{attribute 'linkalways'} 
{attribute 'no_explicit_call' := 'This FB is a CLASS and must be accessed using methods or properties'}
{attribute 'enable_dynamic_creation'}
FUNCTION_BLOCK _GVSP_PIXEL_FORMAT EXTENDS StructuredDatatypeBase
VAR
	localData : GVSP_PIXEL_FORMAT;
	activeData : REFERENCE TO GVSP_PIXEL_FORMAT REF= localData;
    _Color : _BYTE(localdata.Color);
    _EffectivePixelSize : _BYTE(localdata.EffectivePixelSize);
    _Id : _UINT(localdata.Id);
END_VAR

PROPERTY PUBLIC Address : PVOID
GET
Address := ADR(activeData);
END_GET
END_PROPERTY

METHOD PUBLIC ClearReference
VAR_INPUT
END_VAR
activeData REF= localData;
SetMemberReference();
END_METHOD

METHOD PUBLIC Clone : I_Datatype
VAR
    pClone : POINTER TO _GVSP_PIXEL_FORMAT;
END_VAR
pClone := __NEW(_GVSP_PIXEL_FORMAT());
pClone^.Value := Value;
Clone := pClone^;
END_METHOD

PROPERTY PUBLIC Color : REFERENCE TO _BYTE
GET
Color REF= _Color;
END_GET
END_PROPERTY

PROPERTY PUBLIC EffectivePixelSize : REFERENCE TO _BYTE
GET
EffectivePixelSize REF= _EffectivePixelSize;
END_GET
END_PROPERTY

METHOD FB_init : BOOL
VAR_INPUT
	bInitRetains : BOOL; // if TRUE, the retain variables are initialized (warm start / cold start)
	bInCopyCode : BOOL;  // if TRUE, the instance afterwards gets moved into the copy code (online change)
END_VAR
SetMemberReference();
AddMember('Color', _Color);
AddMember('EffectivePixelSize', _EffectivePixelSize);
AddMember('Id', _Id);
END_METHOD

PROPERTY PUBLIC Id : REFERENCE TO _UINT
GET
Id REF= _Id;
END_GET
END_PROPERTY

PROPERTY PUBLIC Identifier : T_MAXSTRING
GET
Identifier := 'GVSP_PIXEL_FORMAT';
END_GET
END_PROPERTY

METHOD PUBLIC MakeReferenceTo
VAR_INPUT
	ReferenceTarget : REFERENCE TO GVSP_PIXEL_FORMAT;
END_VAR
activeData REF= ReferenceTarget;
SetMemberReference();
END_METHOD

METHOD PROTECTED SetMemberReference
VAR_INPUT
END_VAR
_Color.MakeReferenceTo(activeData.Color);
_EffectivePixelSize.MakeReferenceTo(activeData.EffectivePixelSize);
_Id.MakeReferenceTo(activeData.Id);
END_METHOD

PROPERTY PUBLIC Size : UDINT
GET
Size := SIZEOF(activeData);
END_GET
END_PROPERTY

METHOD TryMakeReferenceTo : BOOL
VAR_INPUT
	Target : I_Datatype;
END_VAR
VAR
	targetAsStruct : I_StructuredDatatype;
	pTargetData : POINTER TO GVSP_PIXEL_FORMAT;
END_VAR
IF NOT Target.TryResolveAsStructuredDatatype(targetAsStruct) THEN
	RETURN;
END_IF

IF NOT (targetAsStruct.Identifier = Identifier) THEN
	RETURN;
END_IF

pTargetData := Target.Address;
activeData REF= pTargetData^;
SetMemberReference();
TryMakeReferenceTo := TRUE;
END_METHOD

PROPERTY PUBLIC Value : REFERENCE TO GVSP_PIXEL_FORMAT
GET
Value REF= activeData;
END_GET
END_PROPERTY

END_FUNCTION_BLOCK

(* stored: Version 1.1.0.1, ProductVersion 3.1.4024.13
   POU _GVSP_PIXEL_FORMAT: Id {a116f94a-4213-08f9-1bc6-cc0b5032c34c}, SpecialFunc None
   Folder Core: Id {de03ba50-f102-093f-1e99-918ac2aba4e8}
   Folder Customize: Id {b7f0c839-320c-0814-30bb-2652c18d53f0}
   Folder Constructor: Id {0cf458cc-e85c-0f8c-3bfd-2f71d3f0e86b}
   Folder Protected: Id {3e9643a2-b9e0-0b49-39f0-1d167209cba0}
   Property Address: Id {88409d52-1c3f-0ab2-0db2-91ff5327fa33}
   Get Get: Id {102bb7bb-46d0-0573-006f-553949089485}
   Method ClearReference: Id {076939b8-fec9-0743-1e1a-7befeb74f0ea}
   Method Clone: Id {aceb4875-7f8c-0c8e-1b2a-859d3e372b61}
   Property Color: Id {63f2c747-7a02-009e-1b38-079c669c61fc}
   Get Get: Id {ddb27ea5-cb61-0f11-0c67-4670dba28b88}
   Property EffectivePixelSize: Id {8f567854-4248-0d94-3546-1af57db6f06b}
   Get Get: Id {5c248770-95ff-024a-2754-2bac4a9ffb99}
   Method FB_init: Id {613a00c2-ed3e-06e2-380a-53e95f3b0388}
   Property Id: Id {815ee0ed-97aa-0950-1111-2bf0addaaa0a}
   Get Get: Id {fc816f9a-3861-0c2b-100d-9b4bc7217abd}
   Property Identifier: Id {a4b39483-493e-0295-1bbf-b863fe0fbdae}
   Get Get: Id {b6a39aa2-0101-01e3-19a1-1ca862f6cb9d}
   Method MakeReferenceTo: Id {c0fe64b3-fe65-0dbe-3dcf-a4327ed18531}
   Method SetMemberReference: Id {b2a05782-b3cf-0c2c-0344-579565cd6b6c}
   Property Size: Id {c9c01ad7-8ebc-054b-3f8d-855f0536c0bd}
   Get Get: Id {4d069790-f86d-0d24-3aea-aa299490bc1e}
   Method TryMakeReferenceTo: Id {0c17b3cc-9521-0385-2a18-6b5aea0cb33b}
   Property Value: Id {3a1e4443-0c38-0ca7-1b41-fcbea723e73a}
   Get Get: Id {d66672e0-dab5-0d2a-2936-0867c9be722f} *)
